{attribute 'OPC.UA.DA' := '1'}
TYPE ST_Position :
STRUCT
	x: LREAL; 
	y: LREAL; 
	z: LREAL; 
END_STRUCT
END_TYPE

(* stored: Version 1.1.0.1, ProductVersion 3.1.4024.13
   DUT ST_Position: Id {bed5c334-9297-4de0-9850-d359fb2b8d64} *)
